FUNCTION_BLOCK FB_Filter
VAR_INPUT
	VIn		:	REAL;
END_VAR
VAR_IN_OUT
	VOut	:	REAL;
END_VAR
VAR
	VPrev	:	REAL	:= 0;
	tau		:	REAL	:= 50E-3;
	Tc		:	REAL	:= 10E-3;
	A		:	REAL;
END_VAR

A := tau/(tau + Tc);
VOut  := A*VPrev+(1-A)*VIn;
VPrev := Vout;

END_FUNCTION_BLOCK

(* stored: Version 1.1.0.1, ProductVersion 3.1.4024.12
   POU FB_Filter: Id {bf7ae56e-02d2-445b-a718-de95f7d21e2f}, SpecialFunc None *)
